// LS Electric XG5000 project: 71회예상2_1
// PLC NewPLC
// module base 0 slot 0: 입출력 모듈:XBC-DR20S (DC 24V 입력 12점, 릴레이 출력 8점)

PROGRAM NewProgram (task: 스캔 프로그램)

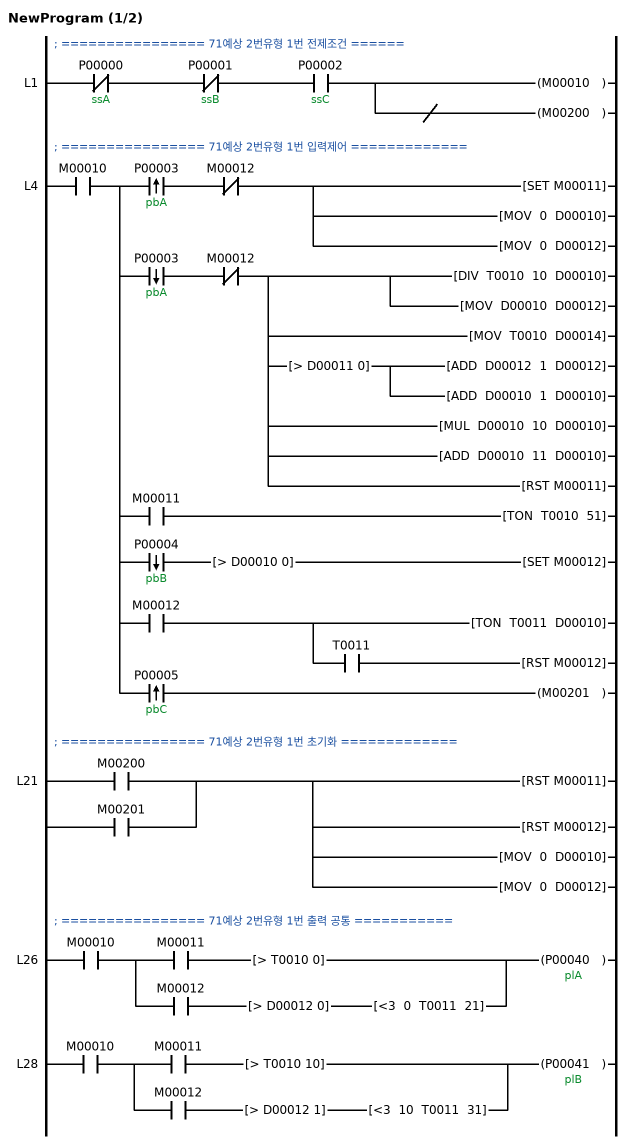
// ================ 71예상 2번유형 1번 전제조건 ======
; L1
LOAD NOT  P00000	// ssA
AND NOT   P00001	// ssB
AND       P00002	// ssC
OUT       M00010
NOT
OUT       M00200
// ================ 71예상 2번유형 1번 입력제어 =============
; L4
LOAD      M00010
MPUSH
ANDP      P00003	// pbA
AND NOT   M00012
SET       M00011
MOV       0 D00010
MOV       0 D00012
MLOAD
ANDN      P00003	// pbA
AND NOT   M00012
DIV       T0010 10 D00010
MOV       D00010 D00012
MOV       T0010 D00014
MPUSH
AND>      D00011 0
ADD       D00012 1 D00012
ADD       D00010 1 D00010
MPOP
MUL       D00010 10 D00010
ADD       D00010 11 D00010
RST       M00011
MLOAD
AND       M00011
TON       T0010 51
MLOAD
ANDN      P00004	// pbB
AND>      D00010 0
SET       M00012
MLOAD
AND       M00012
TON       T0011 D00010
AND       T0011
RST       M00012
MPOP
ANDP      P00005	// pbC
OUT       M00201
// ================ 71예상 2번유형 1번 초기화 =============
; L21
LOAD      M00200
OR        M00201
RST       M00011
RST       M00012
MOV       0 D00010
MOV       0 D00012
// ================ 71예상 2번유형 1번 출력 공통 ===========
; L26
LOAD      M00010
LOAD      M00011
AND>      T0010 0
LOAD      M00012
AND>      D00012 0
AND<3     0 T0011 21
OR LOAD
AND LOAD
OUT       P00040	// plA
; L28
LOAD      M00010
LOAD      M00011
AND>      T0010 10
LOAD      M00012
AND>      D00012 1
AND<3     10 T0011 31
OR LOAD
AND LOAD
OUT       P00041	// plB

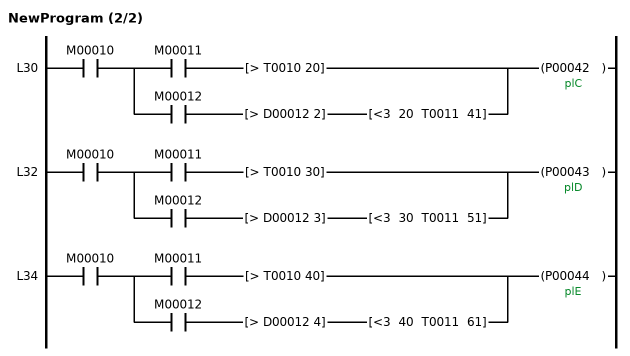
; L30
LOAD      M00010
LOAD      M00011
AND>      T0010 20
LOAD      M00012
AND>      D00012 2
AND<3     20 T0011 41
OR LOAD
AND LOAD
OUT       P00042	// plC
; L32
LOAD      M00010
LOAD      M00011
AND>      T0010 30
LOAD      M00012
AND>      D00012 3
AND<3     30 T0011 51
OR LOAD
AND LOAD
OUT       P00043	// plD
; L34
LOAD      M00010
LOAD      M00011
AND>      T0010 40
LOAD      M00012
AND>      D00012 4
AND<3     40 T0011 61
OR LOAD
AND LOAD
OUT       P00044	// plE